// Mitsubishi GX Works2 project: 14-06-2020 LAB 2   PLC: FX3G

PROGRAM MAIN
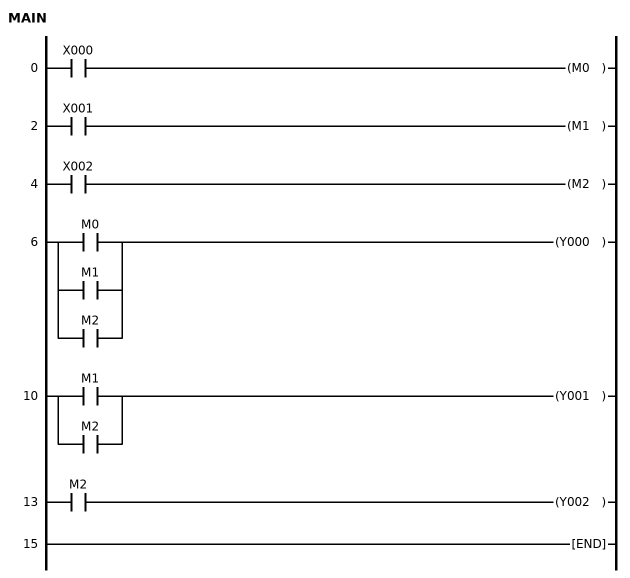
0     LD      X000
      OUT     M0
2     LD      X001
      OUT     M1
4     LD      X002
      OUT     M2
6     LD      M0
      OR      M1
      OR      M2
      OUT     Y000
10    LD      M1
      OR      M2
      OUT     Y001
13    LD      M2
      OUT     Y002
15    END
END_PROGRAM
